Staubli VAL3: save.pgx

public program save(num x_nRetrun)
begin
  x_nRetrun=data:libSave()
end
